# EPICS autosave request: TC/TC_01_settings.req
file "motor_settings.req" P=TE:NDLT1542:, M=MOT:MTR0101
file "motor_settings.req" P=TE:NDLT1542:, M=MOT:MTR0102
file "motor_settings.req" P=TE:NDLT1542:, M=MOT:MTR0103
file "motor_settings.req" P=TE:NDLT1542:, M=MOT:MTR0104
file "motor_settings.req" P=TE:NDLT1542:, M=MOT:MTR0105
file "motor_settings.req" P=TE:NDLT1542:, M=MOT:MTR0106
file "motor_settings.req" P=TE:NDLT1542:, M=MOT:MTR0107
file "motor_settings.req" P=TE:NDLT1542:, M=MOT:MTR0108
file "motor_settings.req" P=TE:NDLT1542:, M=MOT:MTR0109
file "motor_settings.req" P=TE:NDLT1542:, M=MOT:MTR0110
file "motor_settings.req" P=TE:NDLT1542:, M=MOT:MTR0111
